FUNCTION TryConvert_UDINT_TO_DWORD : BOOL
VAR_INPUT
	in : UDINT;
	out : REFERENCE TO DWORD;
END_VAR

out := UDINT_TO_DWORD(in);
TryConvert_UDINT_TO_DWORD := TRUE;

END_FUNCTION

(* stored: Version 1.1.0.1, ProductVersion 3.1.4024.12
   POU TryConvert_UDINT_TO_DWORD: Id {3235d934-f29f-4ba2-b70a-45805e926022}, SpecialFunc None *)
